(* CoDeSys 2.3.9.47 project: ATS_P5_loops.pro *)
(* Libraries: STANDARD.LIB 5.6.98 12:03:02 *)

(* Task configuration *)
TASK Standard (PRIORITY := 0, INTERVAL := T#10ms);
	MAIN
END_TASK

(* POU MAIN, ST *)
PROGRAM MAIN
VAR
(**)
	i_index		: INT;
	i_myArray	: ARRAY [1..10] OF INT;
END_VAR
(*
	Fill Array by FORLOOP
*)
FOR i_index := 1 TO 10 BY 1 DO
    i_myArray[i_index] := i_index*5;
END_FOR;


(*
	Fill Array by WHILELOOP
	(First reset index to one)
*)
i_index := 1;
WHILE i_index <= 10 DO
    i_myArray[i_index] := i_index*3;
	i_index := i_index +1;
END_WHILE;

(*
	Fill Array by REPEAT
	(First reset index to one)
*)
i_index := 1;
REPEAT
	i_myArray[i_index] := i_index;
	i_index := i_index +1;
UNTIL i_index >= 10
END_REPEAT;
END_PROGRAM
